# B&R Automation Studio project lab1_PO
Automation Studio 4.5.2.102

## Configuration Config1

### Task classes (Cpu.sw)
```
Cyclic#4:
  Program <- Program.prg
Libraries: MotCon
```

### Hardware
```
4PP065_0351_P74 : 4PP065.0351-P74 v1.0.4.0
  Connector IF5:
    ActivateDevice = 1
  KeyMappingFile = VC\4PP065_0351_P74.dis
```

## Logical view

### Program Logical/Program (ANSIC)

#### Variables.var
```iecst
VAR
	fb_controller : FB_Regulator;
	Speed : REAL;
	fb_motor : FB_Motor;
	Enable : BOOL;
	fb_motor2 : FB_Motor;
	integrator : FB_Integrator;
	count : REAL;
END_VAR
```

#### Main.c
```c
#include <bur/plctypes.h>

#ifdef _DEFAULT_INCLUDES
	#include <AsDefault.h>
#endif

void _INIT ProgramInit(void)
{
	Enable = 1;
	count = 0;
	Speed = 0;

	fb_motor.dt = 0.01;
	fb_motor.ke = 0.24;
	fb_motor.Tm = 0.1;
	fb_motor.u = 0;
	fb_motor.integrator.dt = 0.01;

	fb_motor2.dt = 0.01;
	fb_motor2.ke = 0.24;
	fb_motor2.Tm = 0.1;
	fb_motor2.u = 0;
	fb_motor2.integrator.dt = 0.01;

	fb_controller.dt = 0.01;
	fb_controller.integrator.dt = 0.01;
	fb_controller.k_i = 7.2*100;
	fb_controller.k_p = 0.24;
	fb_controller.max_abs_value = 24.0;
}

void _CYCLIC ProgramCyclic(void)
{
	if (Enable == 1)
	{
		count += 10;
		if (count >= 500 && count <= 1000) Speed = 40;
		else Speed = 5;
		if (count>1000) count = 0;
	}

	else Speed = 0;
	fb_controller.e = Speed - fb_motor.w;
	fb_motor2.u = Speed * fb_motor2.ke;
	fb_motor.u = fb_controller.u*fb_motor.ke;
	FB_Regulator(&fb_controller);
	FB_Motor(&fb_motor);
	FB_Motor(&fb_motor2);

}

void _EXIT ProgramExit(void)
{

}
```

### Library Logical/MotCon (ANSIC)

#### MotCon.fun - Exported functions and function blocks
```iecst
{REDUND_ERROR} {REDUND_UNREPLICABLE} FUNCTION_BLOCK FB_Integrator (*TODO: Add your comment here*) (*$GROUP=User,$CAT=User,$GROUPICON=User.png,$CATICON=User.png*)
	VAR_INPUT
		in : {REDUND_UNREPLICABLE} REAL;
	END_VAR
	VAR_OUTPUT
		out : {REDUND_UNREPLICABLE} REAL;
	END_VAR
	VAR
		dt : {REDUND_UNREPLICABLE} REAL;
	END_VAR
END_FUNCTION_BLOCK

{REDUND_ERROR} {REDUND_UNREPLICABLE} FUNCTION_BLOCK FB_Motor (*TODO: Add your comment here*) (*$GROUP=User,$CAT=User,$GROUPICON=User.png,$CATICON=User.png*)
	VAR_INPUT
		u : {REDUND_UNREPLICABLE} REAL;
	END_VAR
	VAR_OUTPUT
		w : {REDUND_UNREPLICABLE} REAL;
		phi : {REDUND_UNREPLICABLE} REAL;
	END_VAR
	VAR
		integrator : {REDUND_UNREPLICABLE} FB_Integrator;
		Tm : {REDUND_UNREPLICABLE} REAL;
		ke : {REDUND_UNREPLICABLE} REAL;
		dt : {REDUND_UNREPLICABLE} REAL;
	END_VAR
END_FUNCTION_BLOCK

{REDUND_ERROR} FUNCTION_BLOCK FB_Regulator (*TODO: Add your comment here*) (*$GROUP=User,$CAT=User,$GROUPICON=User.png,$CATICON=User.png*)
	VAR_INPUT
		e : {REDUND_UNREPLICABLE} REAL;
	END_VAR
	VAR_OUTPUT
		u : {REDUND_UNREPLICABLE} REAL;
	END_VAR
	VAR
		k_p : {REDUND_UNREPLICABLE} REAL;
		k_i : {REDUND_UNREPLICABLE} REAL;
		integrator : {REDUND_UNREPLICABLE} FB_Integrator;
		iyOld : {REDUND_UNREPLICABLE} REAL;
		max_abs_value : {REDUND_UNREPLICABLE} REAL;
		dt : {REDUND_UNREPLICABLE} REAL;
		e_p : REAL;
	END_VAR
END_FUNCTION_BLOCK
```

#### FB_Integrator.c
```c
#include <bur/plctypes.h>
#ifdef __cplusplus
	extern "C"
	{
#endif
	#include "MotCon.h"
#ifdef __cplusplus
	};
#endif
/* TODO: Add your comment here */
void FB_Integrator(struct FB_Integrator* inst)
{
	inst->out += inst->in;
}
```

#### FB_Motor.c
```c
#include <bur/plctypes.h>
#ifdef __cplusplus
	extern "C"
	{
#endif
	#include "MotCon.h"
#ifdef __cplusplus
	};
#endif
/* TODO: Add your comment here */
void FB_Motor(struct FB_Motor* inst)
{
	inst->integrator.in = (inst->u*(1/inst->ke) - inst->w)*(inst->dt/inst->Tm);
	FB_Integrator(&(inst->integrator));
	inst->w = inst->integrator.out;
	inst->integrator.in = inst->w*inst->dt;
	FB_Integrator(&(inst->integrator));

	inst->phi = inst->integrator.out;
}
```

#### FB_Regulator.c
```c
#include <bur/plctypes.h>
#ifdef __cplusplus
	extern "C"
	{
#endif
	#include "MotCon.h"
#ifdef __cplusplus
	};
#endif
/* TODO: Add your comment here */
void FB_Regulator(struct FB_Regulator* inst)
{
	inst->integrator.in = inst->e*inst->k_i*inst->dt + inst->iyOld;
	FB_Integrator(&(inst->integrator));
	inst->e_p = inst->e*inst->k_p;
	if (inst->e_p < inst->max_abs_value || inst->e_p > -inst->max_abs_value);
	else
	{
		if (inst->e_p > 0) inst->e_p = inst->max_abs_value;
		else inst->e_p = -inst->max_abs_value;
	}

	inst->e_p += inst->integrator.out;
	if (inst->e_p < inst->max_abs_value || inst->e_p -inst->max_abs_value) inst->u = inst->e_p;
	else
	{
		if (inst->e_p > 0) inst->u = inst->max_abs_value;
		else inst->u = -inst->max_abs_value;
	}
	inst->iyOld = inst->u - inst->e_p;
}
```

Listed in the project but not available here: Logical/Global.typ, Logical/Global.var, Logical/Libraries, Logical/MotCon/Types.typ, Logical/MotCon/Constants.var
